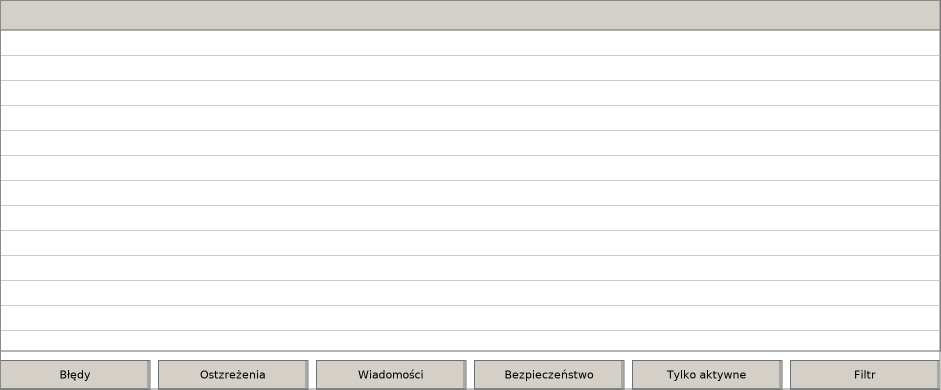
VISUALIZATION Visu_LogowanieBledow_Tabela  // 941x390
VAR_IN_OUT
	stParametry								: DUT_LogowanieBledow_WyswietlanieParametry;
END_VAR
    Table (0,0 941x351), data array: GVL_LogowanieBledow.fbLoger.arrTablicaWyswietlana
        p3854506369: GVL_LogowanieBledow.fbLoger.arrTablicaWyswietlana[INDEX].sNrKomponentu
        p1892666644: GVL_LogowanieBledow.fbLoger.arrTablicaWyswietlana[INDEX].sKodBledu
        p338671338: GVL_LogowanieBledow.fbLoger.arrTablicaWyswietlana[INDEX].byRodzajZdarzenia
        p2170511999: GVL_LogowanieBledow.fbLoger.arrTablicaWyswietlana[INDEX].sOpis
        p3723444502: GVL_LogowanieBledow.fbLoger.arrTablicaWyswietlana[INDEX].dtDataStart
        p1218418051: GVL_LogowanieBledow.fbLoger.arrTablicaWyswietlana[INDEX].dtDataKoniec
        p746581629: GVL_LogowanieBledow.fbLoger.arrTablicaWyswietlana[INDEX].dwKolor
        p2232123230: Nr Elem.
        p2237128397: Data start
        p505689113: Data koniec
        Columns.Column.[3].Template: 16#FF000000 OR (GVL_LogowanieBledow.fbLoger.arrTablicaWyswietlana[INDEX].dwKolor)
    Button (632,360 150x30), "Tylko aktywne", colour toggle: stParametry.bFiltrAktywne
        toggle stParametry.bFiltrAktywne
    Button (0,360 150x30), "Błędy", colour toggle: stParametry.bFiltrRodzaj and stParametry.byFiltrRodzaj = 1
        OnMouseDown: execute {
            (*
            IF (NOT stParametry.bFiltrRodzaj) THEN
            	stParametry.bFiltrRodzaj := TRUE;
            	stParametry.byFiltrRodzaj := 1;
            ELSE
            	stParametry.bFiltrRodzaj := FALSE;
            END_IF
            *)
        }
    Button (158,360 150x30), "Ostzreżenia", colour toggle: stParametry.bFiltrRodzaj and stParametry.byFiltrRodzaj = 2
        OnMouseDown: execute {
            (*
            IF (NOT stParametry.bFiltrRodzaj) THEN
            	stParametry.bFiltrRodzaj := TRUE;
            	stParametry.byFiltrRodzaj := 2;
            ELSE
            	stParametry.bFiltrRodzaj := FALSE;
            END_IF
            *)
        }
    Button (316,360 150x30), "Wiadomości", colour toggle: stParametry.bFiltrRodzaj and stParametry.byFiltrRodzaj = 3
        OnMouseDown: execute {
            (*
            IF (NOT stParametry.bFiltrRodzaj) THEN
            	stParametry.bFiltrRodzaj := TRUE;
            	stParametry.byFiltrRodzaj := 3;
            ELSE
            	stParametry.bFiltrRodzaj := FALSE;
            END_IF
            *)
        }
    Button (474,360 150x30), "Bezpieczeństwo", colour toggle: stParametry.bFiltrRodzaj and stParametry.byFiltrRodzaj = 4
        OnMouseDown: execute {
            (*
            IF (NOT stParametry.bFiltrRodzaj) THEN
            	stParametry.bFiltrRodzaj := TRUE;
            	stParametry.byFiltrRodzaj := 4;
            ELSE
            	stParametry.bFiltrRodzaj := FALSE;
            END_IF
            *)
        }
    Button (790,360 150x30), "Filtr"
END_VISUALIZATION

(* stored: Version 1.1.0.1, ProductVersion 3.1.4024.11
   Visu Visu_LogowanieBledow_Tabela: Id {3dc9ce44-38c3-4cfe-98bb-3fc546ae08da} *)
